// TIA Portal V15.1 program export: 0 tag tables, 0 data types, 0 data blocks, 2 code blocks (in call order from the OBs), 0 instance data blocks

ORGANIZATION_BLOCK "Main"   // OB1, LAD, ProgramCycle
TITLE = "Main Program Sweep (Cycle)"
{ S7_Optimized_Access := 'TRUE' }
// stored: SetENOAutomatically False
   VAR_INPUT
      Initial_Call : Bool;   // Initial call of this OB
      Remanence : Bool;   // =True, if remanent data are available
   END_VAR
BEGIN
END_ORGANIZATION_BLOCK

FUNCTION_BLOCK "块_1"   // FB1, LAD
{ S7_Optimized_Access := 'TRUE' }
// stored: MemoryReserve 100, SetENOAutomatically False
BEGIN
END_FUNCTION_BLOCK
